FUNCTION_BLOCK Visu IMPLEMENTS InterfaceVisu
VAR_INPUT
END_VAR
VAR_OUTPUT
END_VAR
VAR

	//Zustandsautomat
	nZustandsautomatCount		: INT	:= 0;
	VisuSelectedZustandsautomat	: INT := 1;
	VisuNamenZustandsautomaten	: ARRAY[1..KonfigurationVisuZustandsautomat.cMaxZustandsautoamten] 	OF STRING(255);
	VisuPanel					: POINTER TO ST_Panel;
	VisuIpPanel					: ARRAY[1..KonfigurationVisuZustandsautomat.cMaxZustandsautoamten] 	OF POINTER TO ST_Panel;
END_VAR

IF VisuIpPanel[VisuSelectedZustandsautomat] <> 0 THEN
	VisuPanel		:= VisuIpPanel[VisuSelectedZustandsautomat];
END_IF

METHOD ZustandsautomatAddVisu : BOOL
VAR_INPUT
	P_Panel						: POINTER TO ST_Panel;
	Name						: STRING(255);
END_VAR
IF nZustandsautomatCount >= 0
	AND nZustandsautomatCount < KonfigurationVisuZustandsautomat.cMaxZustandsautoamten
THEN
	nZustandsautomatCount := nZustandsautomatCount +1;
	P_Panel^.Name := Name;			
	VisuIpPanel[nZustandsautomatCount] := P_Panel;
	VisuNamenZustandsautomaten[nZustandsautomatCount] := Name;
	ZustandsautomatAddVisu := TRUE;
ELSE
	ZustandsautomatAddVisu := FALSE;
END_IF
END_METHOD

END_FUNCTION_BLOCK

(* stored: Version 1.1.0.1, ProductVersion 3.1.4024.9
   POU Visu: Id {3eca0047-93a4-4746-8e3f-235124f0045c}, SpecialFunc None
   Method ZustandsautomatAddVisu: Id {aacc5658-d565-4e6f-8033-320cc22e6411} *)
